Staubli VAL3: table.dtx

mdesc mNomSpeed
public num nMatrix[1 1]
